TYPE U8 : BYTE; END_TYPE

(* stored: Version 1.1.0.1
   DUT U8: Id {ee03d968-ebc5-0d32-0aef-9fe9085863bf} *)
